FUNCTION_BLOCK PUTTEXT (* openCV text drawer *)
  (* Version 1.0, AN, SWDC RTSoft *)
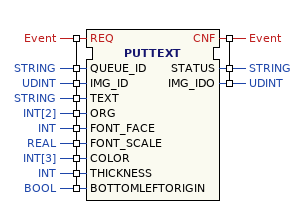
  EVENT_INPUT
    REQ WITH QUEUE_ID, IMG_ID, TEXT, ORG, FONT_FACE, FONT_SCALE, COLOR, THICKNESS, BOTTOMLEFTORIGIN;
  END_EVENT
  EVENT_OUTPUT
    CNF WITH STATUS, IMG_IDO;
  END_EVENT
  VAR_INPUT
    QUEUE_ID : STRING;
    IMG_ID : UDINT;
    TEXT : STRING;
    ORG : ARRAY [0..1] OF INT; (* Bottom-left corner of the text string in the image *)
    FONT_FACE : INT;
    FONT_SCALE : REAL;
    COLOR : ARRAY [0..2] OF INT; (* Color in [B, G, R] *)
    THICKNESS : INT;
    BOTTOMLEFTORIGIN : BOOL; (* When true, the image data origin is at the bottom-left corner, otherwise at the top-left corner *)
  END_VAR
  VAR_OUTPUT
    STATUS : STRING;
    IMG_IDO : UDINT;
  END_VAR
  ALGORITHM REQ IN ST:

  END_ALGORITHM
END_FUNCTION_BLOCK
